FUNCTION_BLOCK AE2_E_TO_EVENT (* Composite FB for convert AE2 to EVENT *)
  (* Standard: 61499-2; Description: Copyright (c) 2024 HR Agrartechnik GmbH This program and the accompanying materials are made available under the terms of the Eclipse Public License 2.0 which is available at https://www.eclipse.org/legal/epl-2.0/ SPDX-License-Identifier: EPL-2.0 *)
  (* Version 1.0, 2024-04-24, Franz Höpfinger, HR Agrartechnik GmbH *)
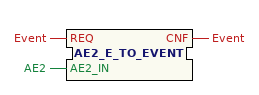
  EVENT_INPUT
    REQ; (* Request to Adapter *)
  END_EVENT
  EVENT_OUTPUT
    CNF; (* Confirmation from Adapter *)
  END_EVENT
  SOCKETS
    AE2_IN : AE2; (* Adapter Input *)
  END_SOCKETS
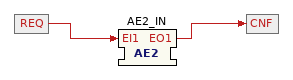
  EVENT_CONNECTIONS
    AE2_IN.EO1 TO CNF;
    REQ TO AE2_IN.EI1;
  END_CONNECTIONS
END_FUNCTION_BLOCK
